(* PLC project tni_train, Dassault Systèmes ControlBuild 2024x *)
(* stored: creationDateTime 2023-10-05T15:44:45-01:00 *)

CONFIGURATION tni_train
  VAR_GLOBAL
    simuperiod : REAL := 50000.0;
    taskname : STRING(50) := 'tni_train.exe';
    allowpreconditions : BOOL := true;
    allowpostconditions : BOOL := true;
    cab1/cabControlPart/keyCabDisabled : BOOL := true;
    cab1/cabControlPart/leftServiceSide : BOOL := true;
    cab2/cabControlPart/keyCabDisabled : BOOL := true;
    cab2/cabControlPart/leftServiceSide : BOOL := true;
  END_VAR
END_CONFIGURATION
